// TwinCAT 3 PLC project Testbench
// Title: Testbench
// Company: Zeugwerk GmbH
// Author: Zeugwerk GmbH
// ProjectVersion: 1.0.0.0
// Description: Lightweight unit-test (adapter) library to be used together with Zeugwerk Creator (Test Explorer)
// ProgramVersion: 3.1.4023.0
// project tree:
//   / IAssertions.TcIO, IUnitTest.TcIO (not stored)

// ---- IAssertions.TcIO
/// Collection of utility methods that support asserting conditions in unittests.
/// The declarations are taken from [TcUnit](https://github.com/tcunit/TcUnit) and the usual implementation
/// of this interface that is used when testing is a wrapper around [FB_TestSuite](https://github.com/tcunit/TcUnit).
/// 
/// For details, see [IUnitTest](xref:Testbench.IUnitTest).
INTERFACE IAssertions

/// Asserts that two objects (of any type) are equal. If they are not, an assertion error is created.
/// For REAL and LREAL it's recommended to use the AssertEquals_REAL or AssertEquals_LREAL respectively
/// as these give the possibility to specify a delta between the expected and actual value.
METHOD PUBLIC Equals
VAR_INPUT
  expected : ANY; //< Expected value
  actual : ANY; //< The value to check against expected
  message : STRING(255); //< The identifying message for the assertion error
END_VAR
END_METHOD

/// Asserts that two LREAL 2D-arrays are equal to within a positive delta. If they are not, an assertion error is created.
METHOD PUBLIC EqualsArray2dLreal
VAR_IN_OUT
  expected : ARRAY[*,*] OF LREAL; //< LREAL 2d array with expected values
  actual : ARRAY[*,*] OF LREAL; //< LREAL 2d array with actual values
END_VAR
VAR_INPUT
  delta : LREAL; //< The maximum delta between the value of expected and actual for which both numbers are still considered equal, proportional to the expected value in that array cell
  message : STRING(255); //< The identifying message for the assertion error
END_VAR
END_METHOD

(*
    Asserts that two REAL 2D-arrays are equal to within a positive delta. If they are not, an assertion error is created.
*)
METHOD PUBLIC EqualsArray2dReal
VAR_IN_OUT
  expected : ARRAY[*,*] OF REAL; //< REAL 2d array with expected values
  actual : ARRAY[*,*] OF REAL; //< REAL 2d array with actual values
END_VAR
VAR_INPUT
  delta : REAL; //< The maximum delta between the value of expected and actual for which both numbers are still considered equal, proportional to the expected value in that array cell
  message : STRING(255); //< The identifying message for the assertion error
END_VAR
END_METHOD

/// Asserts that two LREAL 3D-arrays are equal to within a positive delta. If they are not, an assertion error is created.
METHOD PUBLIC EqualsArray3dLreal
VAR_IN_OUT
  expected : ARRAY[*,*,*] OF LREAL; //< LREAL 3d array with expected values
  actual : ARRAY[*,*,*] OF LREAL; //< LREAL 3d array with actual values
END_VAR
VAR_INPUT
  delta : LREAL; //< The maximum delta between the value of expected and actual for which both numbers are still considered equal, proportional to the expected value in that array cell
  message : STRING(255); //< The identifying message for the assertion error
END_VAR
END_METHOD

/// Asserts that two REAL 3D-arrays are equal to within a positive delta. If they are not, an assertion error is created.
METHOD PUBLIC EqualsArray3dReal
VAR_IN_OUT
  expected : ARRAY[*,*,*] OF REAL; //< REAL 3d array with expected values
  actual : ARRAY[*,*,*] OF REAL; //< REAL 3d array with actual values
END_VAR
VAR_INPUT
  delta : REAL; //< The maximum delta between the value of expected and actual for which both numbers are still considered equal, proportional to the expected value in that array cell
  message : STRING(255); //< The identifying message for the assertion error
END_VAR
END_METHOD

/// Asserts that two BOOL arrays are equal. If they are not, an assertion error is created.
METHOD PUBLIC EqualsArrayBool
VAR_IN_OUT
  expected : ARRAY[*] OF BOOL; //< BOOL array with expected values
  actual : ARRAY[*] OF BOOL; //< BOOL array with actual values
END_VAR
VAR_INPUT
  message : STRING(255); //< The identifying message for the assertion error
END_VAR
END_METHOD

/// Asserts that two BYTE arrays are equal. If they are not, an assertion error is created.
METHOD PUBLIC EqualsArrayByte
VAR_IN_OUT
  expected : ARRAY[*] OF BYTE; //< BYTE array with expected values
  actual : ARRAY[*] OF BYTE; //< BYTE array with actual values
END_VAR
VAR_INPUT
  message : STRING(255); //< The identifying message for the assertion error
END_VAR
END_METHOD

/// Asserts that two DINT arrays are equal. If they are not, an assertion error is created.
METHOD PUBLIC EqualsArrayDint
VAR_IN_OUT
  expected : ARRAY[*] OF DINT; //< DINT array with expected values
  actual : ARRAY[*] OF DINT; //< DINT array with actual values
END_VAR
VAR_INPUT
  message : STRING(255); //< The identifying message for the assertion error
END_VAR
END_METHOD

/// Asserts that two DWORD arrays are equal. If they are not, an assertion error is created.
METHOD PUBLIC EqualsArrayDword
VAR_IN_OUT
  expected : ARRAY[*] OF DWORD; //< DWORD array with expected values
  actual : ARRAY[*] OF DWORD; //< DWORD array with actual values
END_VAR
VAR_INPUT
  message : STRING(255); //< The identifying message for the assertion error
END_VAR
END_METHOD

/// Asserts that two INT arrays are equal. If they are not, an assertion error is created.
METHOD PUBLIC EqualsArrayInt
VAR_IN_OUT
  expected : ARRAY[*] OF INT; //< INT array with expected values
  actual : ARRAY[*] OF INT; //< INT array with actual values
END_VAR
VAR_INPUT
  message : STRING(255); //< The identifying message for the assertion error
END_VAR
END_METHOD

/// Asserts that two LINT arrays are equal. If they are not, an assertion error is created.
METHOD PUBLIC EqualsArrayLint
VAR_IN_OUT
  expected : ARRAY[*] OF LINT; //< LINT array with expected values
  actual : ARRAY[*] OF LINT; //< LINT array with actual values
END_VAR
VAR_INPUT
  message : STRING(255); //< The identifying message for the assertion error
END_VAR
END_METHOD

/// Asserts that two LREAL arrays are equal to within a positive delta. If they are not, an assertion error is created.
METHOD PUBLIC EqualsArrayLreal
VAR_IN_OUT
  expected : ARRAY[*] OF LREAL; //< LREAL array with expected values
  actual : ARRAY[*] OF LREAL; //< LREAL array with actual values
END_VAR
VAR_INPUT
  delta : LREAL; //< The maximum delta between the value of expected and actual for which both numbers are still considered equal, proportional to the expected value in that array cell
  message : STRING(255); //< The identifying message for the assertion error
END_VAR
END_METHOD

/// Asserts that two LWORD arrays are equal. If they are not, an assertion error is created.
METHOD PUBLIC EqualsArrayLword
VAR_IN_OUT
  expected : ARRAY[*] OF LWORD; //< LWORD array with expected values
  actual : ARRAY[*] OF LWORD; //< LWORD array with actual values
END_VAR
VAR_INPUT
  message : STRING(255); //< The identifying message for the assertion error
END_VAR
END_METHOD

/// Asserts that two REAL arrays are equal to within a positive delta. If they are not, an assertion error is created.
METHOD PUBLIC EqualsArrayReal
VAR_IN_OUT
  expected : ARRAY[*] OF REAL; //< REAL array with expected values
  actual : ARRAY[*] OF REAL; //< REAL array with actual values
END_VAR
VAR_INPUT
  delta : REAL; //< The maximum delta between the value of expected and actual for which both numbers are still considered equal, proportional to the expected value in that array cell
  message : STRING(255); //< The identifying message for the assertion error
END_VAR
END_METHOD

/// Asserts that two SINT arrays are equal. If they are not, an assertion error is created.
METHOD PUBLIC EqualsArraySint
VAR_IN_OUT
  expected : ARRAY[*] OF SINT; //< SINT array with expected values
  actual : ARRAY[*] OF SINT; //< SINT array with actual values
END_VAR
VAR_INPUT
  message : STRING(255); //< The identifying message for the assertion error
END_VAR
END_METHOD

/// Asserts that two UDINT arrays are equal. If they are not, an assertion error is created.
METHOD PUBLIC EqualsArrayUdint
VAR_IN_OUT
  expected : ARRAY[*] OF UDINT; //< UDINT array with expected values
  actual : ARRAY[*] OF UDINT; //< UDINT array with actual values
END_VAR
VAR_INPUT
  message : STRING(255); //< The identifying message for the assertion error
END_VAR
END_METHOD

/// Asserts that two UINT arrays are equal. If they are not, an assertion error is created.
METHOD PUBLIC EqualsArrayUint
VAR_IN_OUT
  expected : ARRAY[*] OF UINT; //< UINT array with expected values
  actual : ARRAY[*] OF UINT; //< UINT array with actual values
END_VAR
VAR_INPUT
  message : STRING(255); //< The identifying message for the assertion error
END_VAR
END_METHOD

/// Asserts that two ULINT arrays are equal. If they are not, an assertion error is created.
METHOD PUBLIC EqualsArrayUlint
VAR_IN_OUT
  expected : ARRAY[*] OF ULINT; //< ULINT array with expected values
  actual : ARRAY[*] OF ULINT; //< ULINT array with actual values
END_VAR
VAR_INPUT
  message : STRING(255); //< The identifying message for the assertion error
END_VAR
END_METHOD

/// Asserts that two USINT arrays are equal. If they are not, an assertion error is created.
METHOD PUBLIC EqualsArrayUsint
VAR_IN_OUT
  expected : ARRAY[*] OF USINT; //< USINT array with expected values
  actual : ARRAY[*] OF USINT; //< USINT array with actual values
END_VAR
VAR_INPUT
  message : STRING(255); //< The identifying message for the assertion error
END_VAR
END_METHOD

/// Asserts that two WORD arrays are equal. If they are not, an assertion error is created.
METHOD PUBLIC EqualsArrayWord
VAR_IN_OUT
  expected : ARRAY[*] OF WORD; //< WORD array with expected values
  actual : ARRAY[*] OF WORD; //< WORD array with actual values
END_VAR
VAR_INPUT
  message : STRING(255); //< The identifying message for the assertion error
END_VAR
END_METHOD

/// Asserts that two BOOLs are equal. If they are not, an assertion error is created.
METHOD PUBLIC EqualsBool
VAR_INPUT
  expected : BOOL; //< BOOL expected value
  actual : BOOL; //< BOOL actual value
  message : STRING(255); //< The identifying message for the assertion error
END_VAR
END_METHOD

/// Asserts that two BYTEs are equal. If they are not, an assertion error is created.
METHOD PUBLIC EqualsByte
VAR_INPUT
  expected : BYTE; //< BYTE expected value
  actual : BYTE; //< BYTE actual value
  message : STRING(255); //< The identifying message for the assertion error
END_VAR
END_METHOD

/// Asserts that two DATEs are equal. If they are not, an assertion error is created.
METHOD PUBLIC EqualsDate
VAR_INPUT
  expected : DATE; //< DATE expected value
  actual : DATE; //< DATE actual value
  message : STRING(255); //< The identifying message for the assertion error
END_VAR
END_METHOD

/// Asserts that two DATE_AND_TIMEs are equal. If they are not, an assertion error is created.
METHOD PUBLIC EqualsDateAndTime
VAR_INPUT
  expected : DATE_AND_TIME; //< DATE_AND_TIME expected value
  actual : DATE_AND_TIME; //< DATE_AND_TIME actual value
  message : STRING(255); //< The identifying message for the assertion error
END_VAR
END_METHOD

/// Asserts that two DINTs are equal. If they are not, an assertion error is created.
METHOD PUBLIC EqualsDint
VAR_INPUT
  expected : DINT; //< DINT expected value
  actual : DINT; //< DINT actual value
  message : STRING(255); // The identifying message for the assertion error
END_VAR
END_METHOD

/// Asserts that two DWORDs are equal. If they are not, an assertion error is created.
METHOD PUBLIC EqualsDword
VAR_INPUT
  expected : DWORD; //< DWORD expected value
  actual : DWORD; //< DWORD actual value
  message : STRING(255); //< The identifying message for the assertion error
END_VAR
END_METHOD

/// Asserts that two INTs are equal. If they are not, an assertion error is created.
METHOD PUBLIC EqualsInt
VAR_INPUT
  expected : INT; //< INT expected value
  actual : INT; //< INT actual value
  message : STRING(255); //< The identifying message for the assertion error
END_VAR
END_METHOD

/// Asserts that two LINTs are equal. If they are not, an assertion error is created.
METHOD PUBLIC EqualsLint
VAR_INPUT
  expected : LINT; //< LINT expected value
  actual : LINT; //< LINT actual value
  message : STRING(255); //< The identifying message for the assertion error
END_VAR
END_METHOD

/// Asserts that two LREALs are equal to within a positive delta. If they are not, an assertion error is created.
METHOD PUBLIC EqualsLreal
VAR_INPUT
  expected : LREAL; //< LREAL expected value
  actual : LREAL; //< LREAL actual value
  delta : LREAL; //< The maximum delta between the absolute value of expected and actual for which both numbers are still considered equal
  message : STRING(255); //< The identifying message for the assertion error
END_VAR
END_METHOD

/// Asserts that two LTIMEs are equal. If they are not, an assertion error is created.
METHOD PUBLIC EqualsLtime
VAR_INPUT
  expected : LTIME; //< LTIME expected value
  actual : LTIME; //< LTIME actual value
  message : STRING(255); //< The identifying message for the assertion error
END_VAR
END_METHOD

/// Asserts that two LWORDs are equal. If they are not, an assertion error is created.
METHOD PUBLIC EqualsLword
VAR_INPUT
  expected : LWORD; //< LWORD expected value
  actual : LWORD; //< LWORD actual value
  message : STRING(255); //< The identifying message for the assertion error
END_VAR
END_METHOD

/// Asserts that two REALs are equal to within a positive delta. If they are not, an assertion error is created.
METHOD PUBLIC EqualsReal
VAR_INPUT
  expected : REAL; //< REAL expected value
  actual : REAL; //< REAL actual value
  delta : REAL;  //< The maximum delta between the absolute value of expected and actual for which both numbers are still considered equal
  message : STRING(255); //< The identifying message for the assertion error
END_VAR
END_METHOD

/// Asserts that two SINTs are equal. If they are not, an assertion error is created.
METHOD PUBLIC EqualsSint
VAR_INPUT
  expected : SINT; //< SINT expected value
  actual : SINT; //< SINT actual value
  message : STRING(255); //< The identifying message for the assertion error
END_VAR
END_METHOD

/// Asserts that two STRINGs are equal. If they are not, an assertion error is created.
METHOD PUBLIC EqualsString
VAR_INPUT
  expected : STRING(255); //< STRING expected value
  actual : STRING(255); //< STRING actual value
  message : STRING(255); // The identifying message for the assertion error
END_VAR
END_METHOD

/// Asserts that two TIMEs are equal. If they are not, an assertion error is created.
METHOD PUBLIC EqualsTime
VAR_INPUT
  expected : TIME; //< TIME expected value
  actual : TIME; //< TIME actual value
  message : STRING(255); //< The identifying message for the assertion error
END_VAR
END_METHOD

/// Asserts that two TIME_OF_DAYs are equal. If they are not, an assertion error is created.
METHOD PUBLIC EqualsTimeOfDay
VAR_INPUT
  expected : TIME_OF_DAY; //< TIME_OF_DAY expected value
  actual : TIME_OF_DAY; //< TIME_OF_DAY actual value
  message : STRING(255); //< The identifying message for the assertion error
END_VAR
END_METHOD

/// Asserts that two UDINTs are equal. If they are not, an assertion error is created.
METHOD PUBLIC EqualsUdint
VAR_INPUT
  expected : UDINT; //< UDINT expected value
  actual : UDINT; //< UDINT actual value
  message : STRING(255); //< The identifying message for the assertion error
END_VAR
END_METHOD

/// Asserts that two UINTs are equal. If they are not, an assertion error is created.
METHOD PUBLIC EqualsUint
VAR_INPUT
  expected : UINT; //< UINT expected value
  actual : UINT; //< UINT actual value
  message : STRING(255); //< The identifying message for the assertion error
END_VAR
END_METHOD

/// Asserts that two ULINTs are equal. If they are not, an assertion error is created.
METHOD PUBLIC EqualsUlint
VAR_INPUT
  expected : ULINT; //< ULINT expected value
  actual : ULINT; //< ULINT actual value
  message : STRING(255); //< The identifying message for the assertion error
END_VAR
END_METHOD

/// Asserts that two USINTs are equal. If they are not, an assertion error is created.
METHOD PUBLIC EqualsUsint
VAR_INPUT
  expected : USINT; //< USINT expected value
  actual : USINT; //< USINT actual value
  message : STRING(255); //< The identifying message for the assertion error
END_VAR
END_METHOD

/// Asserts that two WORDs are equal. If they are not, an assertion error is created.
METHOD PUBLIC EqualsWord
VAR_INPUT
  expected : WORD; //< WORD expected value
  actual : WORD; //< WORD actual value
  message : STRING(255); //< The identifying message for the assertion error
END_VAR
END_METHOD

/// Asserts that two WSTRINGs are equal. If they are not, an assertion error is created.
METHOD PUBLIC EqualsWstring
VAR_INPUT
  expected : WSTRING(255); //< WSTRING expected value
  actual : WSTRING(255); //< WSTRING actual value
  message : STRING(255); //< The identifying message for the assertion error
END_VAR
END_METHOD

/// Asserts that a condition is false. If it is not, an assertion error is created.
METHOD PUBLIC IsFalse
VAR_INPUT
  condition : BOOL; //< Condition to be checked
  message : STRING(255); //< The identifying message for the assertion error
END_VAR
END_METHOD

/// Asserts that a condition is true. If it is not, an assertion error is created.
METHOD PUBLIC IsTrue
VAR_INPUT
  condition : BOOL; //< Condition to be checked
  message : STRING(255); //< The identifying message for the assertion error
END_VAR
END_METHOD

END_INTERFACE
